MOVL C09690 V=800.0 PL=0
MOVL C09691 V=800.0 PL=0
MOVL C09692 V=800.0 PL=0
MOVL C09693 V=800.0 PL=0
MOVL C09694 V=800.0 PL=0
MOVL C09695 V=800.0 PL=0
MOVL C09696 V=800.0 PL=0
MOVL C09697 V=800.0 PL=0
MOVL C09698 V=800.0 PL=0
MOVL C09699 V=800.0 PL=0
MOVL C09700 V=800.0 PL=0
MOVL C09701 V=800.0 PL=0
MOVL C09702 V=800.0 PL=0
MOVL C09703 V=800.0 PL=0
MOVL C09704 V=800.0 PL=0
MOVL C09705 V=800.0 PL=0
MOVL C09706 V=800.0 PL=0
MOVL C09707 V=800.0 PL=0
MOVL C09708 V=800.0 PL=0
MOVL C09709 V=800.0 PL=0
MOVL C09710 V=800.0 PL=0
MOVL C09711 V=800.0 PL=0
MOVL C09712 V=800.0 PL=0
MOVL C09713 V=800.0 PL=0
MOVL C09714 V=800.0 PL=0
MOVL C09715 V=800.0 PL=0
MOVL C09716 V=800.0 PL=0
MOVL C09717 V=800.0 PL=0
MOVL C09718 V=800.0 PL=0
MOVL C09719 V=800.0 PL=0
MOVL C09720 V=800.0 PL=0
MOVL C09721 V=800.0 PL=0
MOVL C09722 V=800.0 PL=0
MOVL C09723 V=800.0 PL=0
MOVL C09724 V=800.0 PL=0
MOVL C09725 V=800.0 PL=0
MOVL C09726 V=800.0 PL=0
MOVL C09727 V=800.0 PL=0
MOVL C09728 V=800.0 PL=0
MOVL C09729 V=800.0 PL=0
MOVL C09730 V=800.0 PL=0
MOVL C09731 V=800.0 PL=0
MOVL C09732 V=800.0 PL=0
MOVL C09733 V=800.0 PL=0
MOVL C09734 V=800.0 PL=0
MOVL C09735 V=800.0 PL=0
MOVL C09736 V=800.0 PL=0
MOVL C09737 V=800.0 PL=0
MOVL C09738 V=800.0 PL=0
MOVL C09739 V=800.0 PL=0
MOVL C09740 V=800.0 PL=0
MOVL C09741 V=800.0 PL=0
MOVL C09742 V=800.0 PL=0
MOVL C09743 V=800.0 PL=0
MOVL C09744 V=800.0 PL=0
MOVL C09745 V=800.0 PL=0
MOVL C09746 V=800.0 PL=0
MOVL C09747 V=800.0 PL=0
MOVL C09748 V=800.0 PL=0
MOVL C09749 V=800.0 PL=0
MOVL C09750 V=800.0 PL=0
MOVL C09751 V=800.0 PL=0
MOVL C09752 V=800.0 PL=0
MOVL C09753 V=800.0 PL=0
MOVL C09754 V=800.0 PL=0
MOVL C09755 V=800.0 PL=0
MOVL C09756 V=800.0 PL=0
MOVL C09757 V=800.0 PL=0
MOVL C09758 V=800.0 PL=0
MOVL C09759 V=800.0 PL=0
MOVL C09760 V=800.0 PL=0
MOVL C09761 V=800.0 PL=0
MOVL C09762 V=800.0 PL=0
MOVL C09763 V=800.0 PL=0
MOVL C09764 V=800.0 PL=0
MOVL C09765 V=800.0 PL=0
MOVL C09766 V=800.0 PL=0
MOVL C09767 V=800.0 PL=0
MOVL C09768 V=800.0 PL=0
MOVL C09769 V=800.0 PL=0
MOVL C09770 V=800.0 PL=0
MOVL C09771 V=800.0 PL=0
MOVL C09772 V=800.0 PL=0
MOVL C09773 V=800.0 PL=0
MOVL C09774 V=800.0 PL=0
MOVL C09775 V=800.0 PL=0
MOVL C09776 V=800.0 PL=0
MOVL C09777 V=800.0 PL=0
MOVL C09778 V=800.0 PL=0
MOVL C09779 V=800.0 PL=0
MOVL C09780 V=800.0 PL=0
MOVL C09781 V=800.0 PL=0
MOVL C09782 V=800.0 PL=0
MOVL C09783 V=800.0 PL=0
MOVL C09784 V=800.0 PL=0
MOVL C09785 V=800.0 PL=0
MOVL C09786 V=800.0 PL=0
MOVL C09787 V=800.0 PL=0
MOVL C09788 V=800.0 PL=0
MOVL C09789 V=800.0 PL=0
MOVL C09790 V=800.0 PL=0
MOVL C09791 V=800.0 PL=0
MOVL C09792 V=800.0 PL=0
MOVL C09793 V=800.0 PL=0
MOVL C09794 V=800.0 PL=0
MOVL C09795 V=800.0 PL=0
MOVL C09796 V=800.0 PL=0
MOVL C09797 V=800.0 PL=0
MOVL C09798 V=800.0 PL=0
MOVL C09799 V=800.0 PL=0
MOVL C09800 V=800.0 PL=0
MOVL C09801 V=800.0 PL=0
MOVL C09802 V=800.0 PL=0
MOVL C09803 V=800.0 PL=0
MOVL C09804 V=800.0 PL=0
MOVL C09805 V=800.0 PL=0
MOVL C09806 V=800.0 PL=0
MOVL C09807 V=800.0 PL=0
MOVL C09808 V=800.0 PL=0
MOVL C09809 V=800.0 PL=0
MOVL C09810 V=800.0 PL=0
MOVL C09811 V=800.0 PL=0
MOVL C09812 V=800.0 PL=0
MOVL C09813 V=800.0 PL=0
MOVL C09814 V=800.0 PL=0
MOVL C09815 V=800.0 PL=0
MOVL C09816 V=800.0 PL=0
MOVL C09817 V=800.0 PL=0
MOVL C09818 V=800.0 PL=0
MOVL C09819 V=800.0 PL=0
MOVL C09820 V=800.0 PL=0
MOVL C09821 V=800.0 PL=0
MOVL C09822 V=800.0 PL=0
MOVL C09823 V=800.0 PL=0
MOVL C09824 V=800.0 PL=0
MOVL C09825 V=800.0 PL=0
MOVL C09826 V=800.0 PL=0
MOVL C09827 V=800.0 PL=0
MOVL C09828 V=800.0 PL=0
MOVL C09829 V=800.0 PL=0
MOVL C09830 V=800.0 PL=0
MOVL C09831 V=800.0 PL=0
MOVL C09832 V=800.0 PL=0
MOVL C09833 V=800.0 PL=0
MOVL C09834 V=800.0 PL=0
MOVL C09835 V=800.0 PL=0
MOVL C09836 V=800.0 PL=0
MOVL C09837 V=800.0 PL=0
MOVL C09838 V=800.0 PL=0
MOVL C09839 V=800.0 PL=0
MOVL C09840 V=800.0 PL=0
MOVL C09841 V=800.0 PL=0
MOVL C09842 V=800.0 PL=0
MOVL C09843 V=800.0 PL=0
MOVL C09844 V=800.0 PL=0
MOVL C09845 V=800.0 PL=0
MOVL C09846 V=800.0 PL=0
MOVL C09847 V=800.0 PL=0
MOVL C09848 V=800.0 PL=0
MOVL C09849 V=800.0 PL=0
MOVL C09850 V=800.0 PL=0
MOVL C09851 V=800.0 PL=0
MOVL C09852 V=800.0 PL=0
MOVL C09853 V=800.0 PL=0
MOVL C09854 V=800.0 PL=0
MOVL C09855 V=800.0 PL=0
MOVL C09856 V=800.0 PL=0
MOVL C09857 V=800.0 PL=0
MOVL C09858 V=800.0 PL=0
MOVL C09859 V=800.0 PL=0
MOVL C09860 V=800.0 PL=0
MOVL C09861 V=800.0 PL=0
MOVL C09862 V=800.0 PL=0
MOVL C09863 V=800.0 PL=0
MOVL C09864 V=800.0 PL=0
MOVL C09865 V=800.0 PL=0
MOVL C09866 V=800.0 PL=0
MOVL C09867 V=800.0 PL=0
MOVL C09868 V=800.0 PL=0
MOVL C09869 V=800.0 PL=0
MOVL C09870 V=800.0 PL=0
MOVL C09871 V=800.0 PL=0
MOVL C09872 V=800.0 PL=0
MOVL C09873 V=800.0 PL=0
MOVL C09874 V=800.0 PL=0
MOVL C09875 V=800.0 PL=0
MOVL C09876 V=800.0 PL=0
MOVL C09877 V=800.0 PL=0
MOVL C09878 V=800.0 PL=0
MOVL C09879 V=800.0 PL=0
MOVL C09880 V=800.0 PL=0
MOVL C09881 V=800.0 PL=0
MOVL C09882 V=800.0 PL=0
MOVL C09883 V=800.0 PL=0
MOVL C09884 V=800.0 PL=0
MOVL C09885 V=800.0 PL=0
MOVL C09886 V=800.0 PL=0
MOVL C09887 V=800.0 PL=0
MOVL C09888 V=800.0 PL=0
MOVL C09889 V=800.0 PL=0
MOVL C09890 V=800.0 PL=0
MOVL C09891 V=800.0 PL=0
MOVL C09892 V=800.0 PL=0
MOVL C09893 V=800.0 PL=0
MOVL C09894 V=800.0 PL=0
MOVL C09895 V=800.0 PL=0
MOVL C09896 V=800.0 PL=0
MOVL C09897 V=800.0 PL=0
MOVL C09898 V=800.0 PL=0
MOVL C09899 V=800.0 PL=0
MOVL C09900 V=800.0 PL=0
MOVL C09901 V=800.0 PL=0
MOVL C09902 V=800.0 PL=0
MOVL C09903 V=800.0 PL=0
MOVL C09904 V=800.0 PL=0
MOVL C09905 V=800.0 PL=0
MOVL C09906 V=800.0 PL=0
MOVL C09907 V=800.0 PL=0
MOVL C09908 V=800.0 PL=0
MOVL C09909 V=800.0 PL=0
MOVL C09910 V=800.0 PL=0
MOVL C09911 V=800.0 PL=0
MOVL C09912 V=800.0 PL=0
MOVL C09913 V=800.0 PL=0
MOVL C09914 V=800.0 PL=0
MOVL C09915 V=800.0 PL=0
MOVL C09916 V=800.0 PL=0
MOVL C09917 V=800.0 PL=0
MOVL C09918 V=800.0 PL=0
MOVL C09919 V=800.0 PL=0
MOVL C09920 V=800.0 PL=0
MOVL C09921 V=800.0 PL=0
MOVL C09922 V=800.0 PL=0
MOVL C09923 V=800.0 PL=0
MOVL C09924 V=800.0 PL=0
MOVL C09925 V=800.0 PL=0
MOVL C09926 V=800.0 PL=0
MOVL C09927 V=800.0 PL=0
MOVL C09928 V=800.0 PL=0
MOVL C09929 V=800.0 PL=0
MOVL C09930 V=800.0 PL=0
MOVL C09931 V=800.0 PL=0
MOVL C09932 V=800.0 PL=0
MOVL C09933 V=800.0 PL=0
MOVL C09934 V=800.0 PL=0
MOVL C09935 V=800.0 PL=0
MOVL C09936 V=800.0 PL=0
MOVL C09937 V=800.0 PL=0
MOVL C09938 V=800.0 PL=0
MOVL C09939 V=800.0 PL=0
MOVL C09940 V=800.0 PL=0
MOVL C09941 V=800.0 PL=0
MOVL C09942 V=800.0 PL=0
MOVL C09943 V=800.0 PL=0
MOVL C09944 V=800.0 PL=0
MOVL C09945 V=800.0 PL=0
MOVL C09946 V=800.0 PL=0
MOVL C09947 V=800.0 PL=0
MOVL C09948 V=800.0 PL=0
MOVL C09949 V=800.0 PL=0
MOVL C09950 V=800.0 PL=0
MOVL C09951 V=800.0 PL=0
MOVL C09952 V=800.0 PL=0
MOVL C09953 V=800.0 PL=0
MOVL C09954 V=800.0 PL=0
MOVL C09955 V=800.0 PL=0
MOVL C09956 V=800.0 PL=0
MOVL C09957 V=800.0 PL=0
MOVL C09958 V=800.0 PL=0
MOVL C09959 V=800.0 PL=0
MOVL C09960 V=800.0 PL=0
MOVL C09961 V=800.0 PL=0
MOVL C09962 V=800.0 PL=0
MOVL C09963 V=800.0 PL=0
MOVL C09964 V=800.0 PL=0
MOVL C09965 V=800.0 PL=0
MOVL C09966 V=800.0 PL=0
MOVL C09967 V=800.0 PL=0
MOVL C09968 V=800.0 PL=0
MOVL C09969 V=800.0 PL=0
MOVL C09970 V=800.0 PL=0
MOVL C09971 V=800.0 PL=0
MOVL C09972 V=800.0 PL=0
MOVL C09973 V=800.0 PL=0
MOVL C09974 V=800.0 PL=0
MOVL C09975 V=800.0 PL=0
MOVL C09976 V=800.0 PL=0
MOVL C09977 V=800.0 PL=0
MOVL C09978 V=800.0 PL=0
MOVL C09979 V=800.0 PL=0
MOVL C09980 V=800.0 PL=0
MOVL C09981 V=800.0 PL=0
MOVL C09982 V=800.0 PL=0
MOVL C09983 V=800.0 PL=0
MOVL C09984 V=800.0 PL=0
MOVL C09985 V=800.0 PL=0
MOVL C09986 V=800.0 PL=0
MOVL C09987 V=800.0 PL=0
MOVL C09988 V=800.0 PL=0
MOVL C09989 V=800.0 PL=0
MOVL C09990 V=800.0 PL=0
MOVL C09991 V=800.0 PL=0
MOVL C09992 V=800.0 PL=0
MOVL C09993 V=800.0 PL=0
MOVL C09994 V=800.0 PL=0
MOVL C09995 V=800.0 PL=0
MOVL C09996 V=800.0 PL=0
CALL JOB:A_NAIHAN_0617_1_PAINT_3
END
